ABB RAPID module: MainR.mod

MODULE MainR

    PERS robtarget CupGrid{8};
    PERS bool CupGridFull{8};

    PROC main()


    ENDPROC



ENDMODULE
